PROGRAM SecondPouCreatedFromUser1
VAR
END_VAR

END_PROGRAM

(* stored: Version 1.1.0.1
   POU SecondPouCreatedFromUser1: Id {23c9bc51-90da-48f5-9c99-1434c8e1270a}, SpecialFunc None *)
